SUBAPPLICATION Uebung_003a (* DigitalInput_I1/_I2 auf DigitalOutput_Q1/_I2 *)
  (* Standard: 61499-2 *)
  (* Version 1.0, 2023-10-23, franz *)
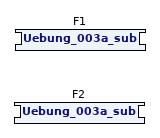
  SUBAPPS
    F1 : Uebung_003a_sub;
    F2 : Uebung_003a_sub;
  END_SUBAPPS
END_SUBAPPLICATION
